SUBAPPLICATION Uebung_003e (* DigitalInput_I1-4 auf DigitalOutput_Q1-4 - flach mit Bypass (Druckumlaufventil) *)
  (* Standard: 61499-2; Description: Copyright (c) 2023 Meisterschulen am Ostbahnhof This program and the accompanying materials are made available under the terms of the Eclipse Public License 2.0 which is available at https://www.eclipse.org/legal/epl-2.0/ SPDX-License-Identifier: EPL-2.0 *)
  (* Version 1.0, 2023-10-23, Franz Höpfinger, Meisterschulen am Ostbahnhof, initial API and implementation and/or initial documentation *)
  PACKAGE Uebungen;
  IMPORT logiBUS::io::DI::logiBUS_DI::Input_I1;
  IMPORT logiBUS::io::DI::logiBUS_DI::Input_I2;
  IMPORT logiBUS::io::DI::logiBUS_DI::Input_I3;
  IMPORT logiBUS::io::DI::logiBUS_DI::Input_I4;
  IMPORT logiBUS::io::DQ::logiBUS_DO::Output_Q1;
  IMPORT logiBUS::io::DQ::logiBUS_DO::Output_Q2;
  IMPORT logiBUS::io::DQ::logiBUS_DO::Output_Q3;
  IMPORT logiBUS::io::DQ::logiBUS_DO::Output_Q4;
  IMPORT logiBUS::io::DQ::logiBUS_DO::Output_Q8;
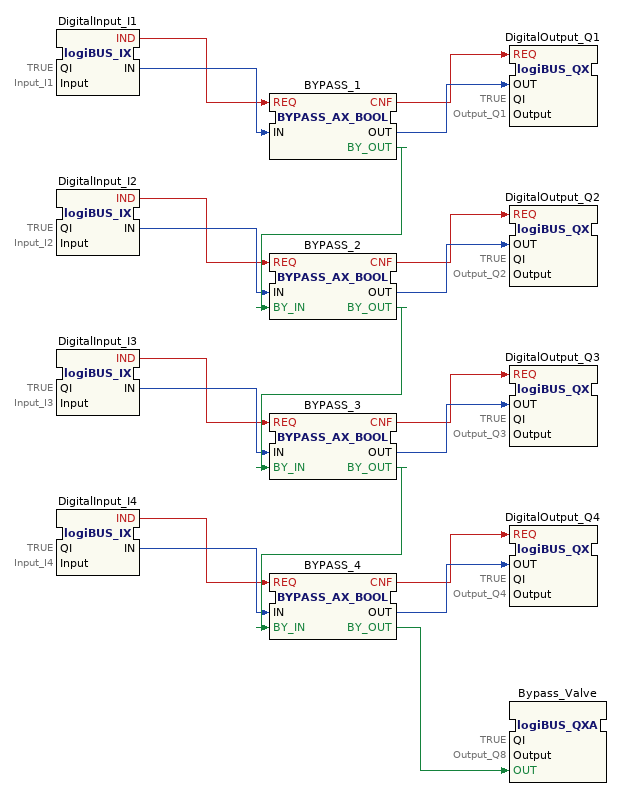
  FBS
    DigitalOutput_Q1 : logiBUS::io::DQ::logiBUS_QX(QI := TRUE, Output := Output_Q1);
    DigitalInput_I1 : logiBUS::io::DI::logiBUS_IX(QI := TRUE, Input := Input_I1);
    DigitalOutput_Q2 : logiBUS::io::DQ::logiBUS_QX(QI := TRUE, Output := Output_Q2);
    DigitalInput_I2 : logiBUS::io::DI::logiBUS_IX(QI := TRUE, Input := Input_I2);
    BYPASS_1 : logiBUS::signalprocessing::bypass::BYPASS_AX_BOOL;
    Bypass_Valve : logiBUS::io::DQ::logiBUS_QXA(QI := TRUE, Output := Output_Q8);
    BYPASS_2 : logiBUS::signalprocessing::bypass::BYPASS_AX_BOOL;
    DigitalOutput_Q3 : logiBUS::io::DQ::logiBUS_QX(QI := TRUE, Output := Output_Q3);
    DigitalInput_I3 : logiBUS::io::DI::logiBUS_IX(QI := TRUE, Input := Input_I3);
    BYPASS_3 : logiBUS::signalprocessing::bypass::BYPASS_AX_BOOL;
    DigitalOutput_Q4 : logiBUS::io::DQ::logiBUS_QX(QI := TRUE, Output := Output_Q4);
    DigitalInput_I4 : logiBUS::io::DI::logiBUS_IX(QI := TRUE, Input := Input_I4);
    BYPASS_4 : logiBUS::signalprocessing::bypass::BYPASS_AX_BOOL;
  END_FBS
  EVENT_CONNECTIONS
    DigitalInput_I1.IND TO BYPASS_1.REQ;
    BYPASS_1.CNF TO DigitalOutput_Q1.REQ;
    DigitalInput_I2.IND TO BYPASS_2.REQ;
    BYPASS_2.CNF TO DigitalOutput_Q2.REQ;
    DigitalInput_I3.IND TO BYPASS_3.REQ;
    BYPASS_3.CNF TO DigitalOutput_Q3.REQ;
    DigitalInput_I4.IND TO BYPASS_4.REQ;
    BYPASS_4.CNF TO DigitalOutput_Q4.REQ;
  END_CONNECTIONS
  DATA_CONNECTIONS
    DigitalInput_I1.IN TO BYPASS_1.IN;
    BYPASS_1.OUT TO DigitalOutput_Q1.OUT;
    DigitalInput_I2.IN TO BYPASS_2.IN;
    BYPASS_2.OUT TO DigitalOutput_Q2.OUT;
    DigitalInput_I3.IN TO BYPASS_3.IN;
    BYPASS_3.OUT TO DigitalOutput_Q3.OUT;
    DigitalInput_I4.IN TO BYPASS_4.IN;
    BYPASS_4.OUT TO DigitalOutput_Q4.OUT;
  END_CONNECTIONS
  ADAPTER_CONNECTIONS
    BYPASS_1.BY_OUT TO BYPASS_2.BY_IN;
    BYPASS_2.BY_OUT TO BYPASS_3.BY_IN;
    BYPASS_3.BY_OUT TO BYPASS_4.BY_IN;
    BYPASS_4.BY_OUT TO Bypass_Valve.OUT;
  END_CONNECTIONS
END_SUBAPPLICATION
